FUNCTION_BLOCK FB_ControlBox
VAR_INPUT
	bRealControlBox : BOOL;
END_VAR
VAR_OUTPUT
	eMode : E_Control_Mode;
	eStatus : E_Status;
END_VAR
VAR
	fbVirtualControlBox : FB_Virtual_Controller;
	fbRealControlBox : FB_Real_Controller;
	fbSelectedControlBox : I_ControlBox := fbVirtualControlBox;
END_VAR

IF bRealControlBox THEN
	fbSelectedControlBox := fbRealControlBox;
ELSE
	fbVirtualControlBox.Lamps();
END_IF

fbSelectedControlBox.Mode(eMode => eMode);
fbSelectedControlBox.Status(eStatus => eStatus);

END_FUNCTION_BLOCK

(* stored: Version 1.1.0.1, ProductVersion 3.1.4024.12
   POU FB_ControlBox: Id {4cfcb7b4-a156-4619-af4f-632ef49bc277}, SpecialFunc None *)
